(* PLC project Example, Beckhoff Automation GmbH TwinCAT PLC Control 3.5.13.20 *)
(* stored: creationDateTime 2020-07-07T10:35:37.2985488, modificationDateTime 2020-07-07T10:35:37.3005449 *)

PROGRAM Example
VAR
	A: BOOL;
	B: BOOL;
END_VAR

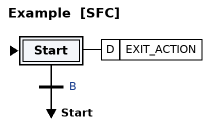
INITIAL_STEP Start:
  EXIT_ACTION(D);
END_STEP
TRANSITION FROM Start TO Start
  := B;
END_TRANSITION

ACTION EXIT_ACTION:
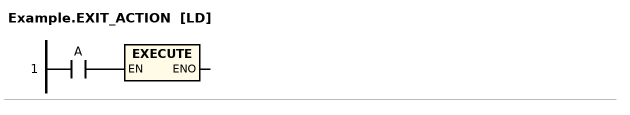
(* LD diagram, written out as Structured Text *)

IF A THEN
  IF A THEN
  	B:= FALSE;
  END_IF
END_IF;
END_ACTION
END_PROGRAM

CONFIGURATION Application
  RESOURCE Example ON PLC
    TASK PlcTask(INTERVAL := T#0ms, PRIORITY := 20);
    PROGRAM MAIN WITH PlcTask : MAIN;
  END_RESOURCE
END_CONFIGURATION
